INTERFACE I_GENERAL

METHOD M_CyclicRun : BOOL
VAR_INPUT
END_VAR
END_METHOD

PROPERTY P_ObjectID : STRING
GET
END_GET
SET
END_SET
END_PROPERTY

END_INTERFACE

(* stored: Version 1.1.0.1, ProductVersion 3.1.4024.12
   Itf I_GENERAL: Id {b877ffd7-cb87-4368-8804-41aa5666923a}
   Method M_CyclicRun: Id {4e304cb9-56de-449c-b8c1-8ab8fbc31ed6}
   Property P_ObjectID: Id {30d6b7eb-5934-4807-bff4-c5c7e206c07a}
   Get Get: Id {7c1c1e94-1dc8-4e93-bbf8-9fb0399fd038}
   Set Set: Id {fc2501e5-c238-487d-a54d-06445a3fec3e} *)
